// TIA Portal V20 export
TYPE "typeFDoorFunction"
// Safety status of door
// stored: Access Published, IsFailsafeCompliant true, Namespace Safety
   STRUCT
      fDoor1 { S7_SetPoint := 'True'} : "Safety.typeFDoorFunctionData";
      fDoor2 { S7_SetPoint := 'True'} : "Safety.typeFDoorFunctionData";
      fDoor3 { S7_SetPoint := 'True'} : "Safety.typeFDoorFunctionData";
      fDoor4 { S7_SetPoint := 'True'} : "Safety.typeFDoorFunctionData";
      fDoor5 { S7_SetPoint := 'True'} : "Safety.typeFDoorFunctionData";
      fDoor6 { S7_SetPoint := 'True'} : "Safety.typeFDoorFunctionData";
      fDoor7 { S7_SetPoint := 'True'} : "Safety.typeFDoorFunctionData";
   END_STRUCT;
END_TYPE
